PROGRAM MAIN
VAR
	fbMotor: fbAbsolute;
	
	fbPower		:mc_Power;
	fbAbsolute  :mc_MoveAbsolute;
	axis		:axis_ref;
	
	ftrboEnable	:f_trig;
END_VAR


gvl.stData.lrActualPos:=axis.NcToPlc.ActPos;
gvl.stData.lrActualVelo:=axis.NcToPlc.ActVelo;
gvl.stData.lrActualAcc:=axis.NcToPlc.ActAcc;

fbMotor(
	boEnable:=gvl.stData.boEnable , 
	boStart:=gvl.stData.boStart , 
	lrPos:=gvl.stData.lrPosition , 
	lrVelo:=gvl.stData.lrVelocity , 
	lrAcc:=gvl.stData.lrAcceleration , 
	lrDec:=gvl.stData.lrDeceleration , 
	lrJerk:=gvl.stData.lrJerk , 
	fbPower:=fbPower , 
	fbAbsolute:=fbAbsolute , 
	axis:=axis );
	
IF fbAbsolute.Done THEN
	gvl.stData.boStart:=false;
END_IF 

ftrboEnable(CLK:=gvl.stData.boEnable);

IF ftrboEnable.Q THEN
	gvl.stData.boStart:=false;
END_IF

END_PROGRAM

(* stored: Version 1.1.0.1, ProductVersion 3.1.4024.12
   POU MAIN: Id {7c126c04-4e7f-4582-b806-5142ed89f896}, SpecialFunc None *)
